Fanuc KAREL source: kt00183.KL

-- PROVISIONAL review KL for V1013-1; original PC SHA256 c7d516df41a61a6b038394630bb7e72e9495c7d962214cf66112baecfa1b698a
-- Incomplete behavior may be omitted. Consult companion uncertainty JSON. Do not deploy.
PROGRAM KT00183
%NOLOCKGROUP
VAR
  OUT : INTEGER
-- UNRESOLVED_DECL Y1 type=002018
-- UNRESOLVED_DECL H2 type=002017
BEGIN
  -- UNRESOLVED_PC offsets 5-19; opcodes 2E,22,9D,33,B2
  -- UNRESOLVED_PC offsets 24-38; opcodes 2E,22,9D,33,B4
  -- UNRESOLVED_PC offsets 43-68; opcodes 22,9D,33,B1,22,9D,33,B3,56,23
  -- UNRESOLVED_PC offsets 73-77; opcodes 7F
END KT00183
